// TIA Portal V18 export
DATA_BLOCK "Pid Control A"   // DB311
{ S7_Optimized_Access := 'TRUE' }
VERSION : 0.1
// stored: AutoNumber false, DBAccessibleFromOPCUA true, IsOnlyStoredInLoadMemory false, IsRetainMemResEnabled false, IsWriteProtectedInAS false, MemoryReserve 100
   VAR
      input : Struct
         setflowrate : Real;
         "Flowrate input" : Real;
         "current flowrate" : Real;
         "Ramp up rate" : Real;
         start : Bool;
         "delay time On" : Bool;
         "setflowrate Low" : Real;
         "setflowrate high" : Real;
         "output low" : Real;
         "output high" : Real;
         "input low" : Real;
         "input high" : Real;
      END_STRUCT;
   END_VAR
   VAR RETAIN
      Control : Struct
         P : Real;
         i : Real;
         d : Real;
         "rampup time" : Real;
         "Activate manual mode" : Bool;
         "Start Delay time" : DInt;
      END_STRUCT;
   END_VAR
   VAR
      Output : Struct
         "output percentage" : Real;
      END_STRUCT;
      Misc : Struct
         error : Bool;
         "error bits" : Int;
         states : Int;
      END_STRUCT;
   END_VAR
   VAR RETAIN
      Enable : Int;
   END_VAR
BEGIN
END_DATA_BLOCK
